FUNCTION_BLOCK DiagServer1 (* Sends sensor data and diagnostic data over a network upon reques. Wrapper for a SERVER function block. *)
  (* Standard: 61499-2; Description: A client can request measurements and diagnostic data from this function block. Requests should be made in regular intervals according to the data input DT. *)
  (* Version 1.0, 2017-08-27, Marc Jakobi, HTW Berlin *)
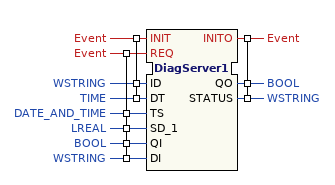
  EVENT_INPUT
    INIT WITH ID, DT; (* Initialization Request *)
    REQ WITH SD_1, DI, QI, TS; (* Normal Execution Request *)
  END_EVENT
  EVENT_OUTPUT
    INITO WITH QO, STATUS; (* Initialization Confirm *)
  END_EVENT
  VAR_INPUT
    ID : WSTRING; (* Connection identifier *)
    DT : TIME := T#1m; (* Client request interval *)
    TS : DATE_AND_TIME; (* Time stamp *)
    SD_1 : LREAL; (* Input data *)
    QI : BOOL; (* Diagnostic qualifier *)
    DI : WSTRING; (* Diagnostic info *)
  END_VAR
  VAR_OUTPUT
    QO : BOOL; (* Output event qualifier *)
    STATUS : WSTRING; (* Service status *)
  END_VAR
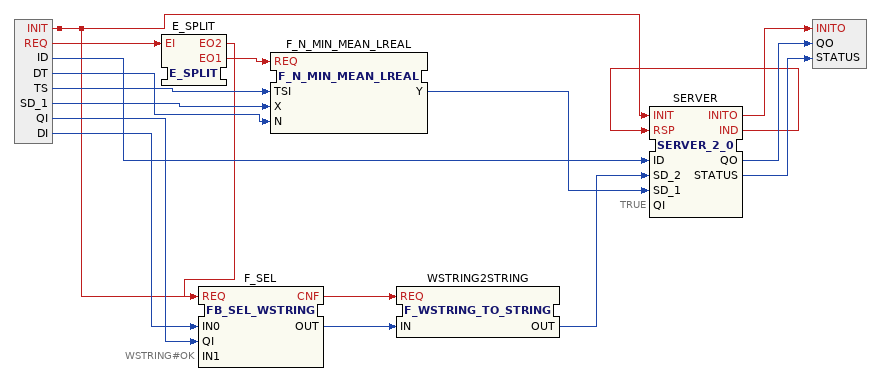
  FBS
    WSTRING2STRING : F_WSTRING_TO_STRING;
    SERVER : SERVER_2_0(QI := TRUE);
    F_SEL : FB_SEL_WSTRING(IN1 := WSTRING#OK);
    F_N_MIN_MEAN_LREAL : F_N_MIN_MEAN_LREAL;
    E_SPLIT : E_SPLIT;
  END_FBS
  EVENT_CONNECTIONS
    INIT TO SERVER.INIT;
    SERVER.INITO TO INITO;
    INIT TO F_SEL.REQ;
    F_SEL.CNF TO WSTRING2STRING.REQ;
    SERVER.IND TO SERVER.RSP;
    REQ TO E_SPLIT.EI;
    E_SPLIT.EO2 TO F_SEL.REQ;
    E_SPLIT.EO1 TO F_N_MIN_MEAN_LREAL.REQ;
  END_CONNECTIONS
  DATA_CONNECTIONS
    ID TO SERVER.ID;
    WSTRING2STRING.OUT TO SERVER.SD_2;
    SERVER.QO TO QO;
    SERVER.STATUS TO STATUS;
    DI TO F_SEL.IN0;
    F_SEL.OUT TO WSTRING2STRING.IN;
    QI TO F_SEL.QI;
    TS TO F_N_MIN_MEAN_LREAL.TSI;
    SD_1 TO F_N_MIN_MEAN_LREAL.X;
    DT TO F_N_MIN_MEAN_LREAL.N;
    F_N_MIN_MEAN_LREAL.Y TO SERVER.SD_1;
  END_CONNECTIONS
END_FUNCTION_BLOCK
